# EPICS substitutions: viocs/tb_ps/tb_psApp/Db/quad.substitutions
file "db/individual.db" {
    pattern { family, pos }
        { "Q1A", "01-A"}
        { "Q1A", "01-B"}
        { "Q1B", "01"}
        { "Q1C", "01"}
        { "QD", "02"}
        { "QF", "02"}
        { "QD", "03-A"}
        { "QF", "03-A"}
        { "QF", "03-B"}
        { "QD", "03-B"}
        { "QF", "04"}
        { "QD", "04"}
        { "QF", "05"}
        { "QD", "05"}
}
